INTERFACE I_NodeFactoryCollection

METHOD PUBLIC GetByType : I_NodeFactory
VAR_INPUT
	NodeType : T_MAXSTRING;
END_VAR
END_METHOD

METHOD PUBLIC HasType : BOOL
VAR_INPUT
	NodeType : T_MAXSTRING;
END_VAR
END_METHOD

METHOD PUBLIC InsertByType
VAR_INPUT
	NodeType : T_MAXSTRING;
	NodeFactory : I_NodeFactory;
END_VAR
END_METHOD

END_INTERFACE

(* stored: Version 1.1.0.1, ProductVersion 3.1.4024.12
   Itf I_NodeFactoryCollection: Id {dd179a1b-4888-0e12-32c8-17e1500648bc}
   Method GetByType: Id {9fba0aae-689e-0867-1abf-4a0a90b87cb8}
   Method HasType: Id {054a4636-e86d-0de8-2332-932e11d4c024}
   Method InsertByType: Id {0a11f8bd-8007-07b8-0f00-2dc2647d18ae} *)
